Staubli VAL3: CartesianAccel.dtx

public num ax
public num ay
public num az
public num arx
public num ary
public num arz
